// TIA Portal V17 export
// export: Created 2025-03-10T13:11:22.6633057Z, ExportSetting WithDefaults, DisplayName Totally Integrated Automation Portal, DisplayVersion V17 Update 8, DisplayName TIA Portal Openness, DisplayVersion V17 Update 8, DisplayName TIA Portal Version Control Interface, DisplayVersion V17, DisplayName SINAMICS Startdrive Advanced, DisplayVersion V17 SP2, DisplayName SINAMICS Startdrive G110M, G120, G120C, G120D, G120P, G115D, DisplayVersion V17 SP2, DisplayName SINAMICS Startdrive G130, G150, S120, S150, SINAMICS MV, S210, DisplayVersion V17 SP2, DisplayName STEP 7 Professional, DisplayVersion V17 Update 8, DisplayName SINUMERIK ONE STEP 7 Toolbox, DisplayVersion V17 Update 12, DisplayName SINUMERIK 840D sl STEP 7 Toolbox, DisplayVersion V17 Update 12, DisplayName STEP 7 Safety, DisplayVersion V17 Update 6, DisplayName WinCC Advanced, DisplayVersion V17 Update 8
FUNCTION_BLOCK "FB6600_SAFETY_BRAKE_Z_AXIS"   // FB6600, LAD
{ S7_Optimized_Access := 'FALSE' }
AUTHOR : ETXETAR
VERSION : 1.0
// stored: AutoNumber false, IsIECCheckEnabled false, SetENOAutomatically false, UDAEnableTagReadback false
   VAR_INPUT
      OPTIONS_0 : Byte := 2#0000_0000;   // OPTION
      BLOCKED_1 : Bool;   // BLOCKED INPUT
      UNBLOCKED_1 : Bool;   // UNBLOCKED INPUT
      MAINT_BLOCKED : Bool;   // MAINTENANCE BLOCKED INPUT
      MAINT_UNBLOCKED : Bool;   // MAINTENANCE UNBLOCKED INPUT
      BLOCK_CONDITIONS : Bool;   // BLOCK CONDITIONS INPUT
      UNBLOCK_CONDITIONS : Bool;   // UNBLOCK CONDITIONS INPUT
      AXIS_SELECTED : Bool;   // AXES SCREEN AXIS SELECTED
      TRAVERSE_COMMAND : Bool;   // TRAVERSE COMMAND FOR THE AXIS
      UNBLOCK_MAN_REQUEST : Bool;   // UNBLOCK MANUAL REQUEST
      BLOCK_AUTO_REQUEST : Bool;   // BLOCK AUTO REQUEST
      UNBLOCK_AUTO_REQUEST : Bool;   // UNBLOCK AUTO REQUEST
      BRAKE_TEST : Bool;   // BRAKE TEST SIGNAL OF THE AXIS
      UNIT_ALARM : UInt;   // UNIT NUMBER MAX. NUMBER=10
      STATION_ALARM : UInt;   // UNIT NUMBER MAX. NUMBER=10
   END_VAR
   VAR_OUTPUT
      BLOCKED : Bool;   // BLOCKED
      UNBLOCKED : Bool;   // UNBLOCKED
      BLOCKED_ALARM : Bool;   // BLOCKED ALARM
      UNBLOCKED_ALARM : Bool;   // UNBLOCKED ALARM
      MAINTENANCE_UNBLOCKED_ALARM : Bool;   // MAINTENANCE UNBLOCKED ALARM
      BLOCK : Bool;   // BLOCK
      UNBLOCK : Bool;   // UNBLOCK
   END_VAR
   VAR DB_SPECIFIC
      BRAKE { S7_SetPoint := 'True'} : "SAFETY_BRAKE";
      TIMER_BLOCKED { S7_SetPoint := 'True'} : TON_TIME;   // BLOCKED TIMER
      TIMER_UNBLOCKED { S7_SetPoint := 'True'} : TON_TIME;   // UNBLOCKED TIMER
      TIMER_SIMULTANEITY { S7_SetPoint := 'True'} : TON_TIME;   // SIMULTANEITY TIMER
      TIMER_TIME_EXCEEDED { S7_SetPoint := 'True'} : TON_TIME;   // TIME EXCEEDED TIMER
   END_VAR
   VAR_TEMP
      INPUTS_MASK : Byte;   // INPUT MASK
      O_BYTE_0 : Struct   // OPTIONS BYTE 0
         MAINTENANCE_SENSORS : Bool;   // MAINTENANCE SENSORS OPTION
         SPARE_1 : Bool;   // SPARE OPTION
         SPARE_2 : Bool;   // SPARE OPTION
         SPARE_3 : Bool;   // SPARE OPTION
         SPARE_4 : Bool;   // SPARE OPTION
         SPARE_5 : Bool;   // SPARE OPTION
         SPARE_6 : Bool;   // SPARE OPTION
         SPARE_7 : Bool;   // SPARE OPTION
      END_STRUCT;
      DB_NUMBER : DInt;   // DB NUMBER FOR ALARM AND HELP DECODING
   END_VAR
   // TIMER_BLOCKED.PT := T#200ms;
   // TIMER_UNBLOCKED.PT := T#150ms;
   // TIMER_SIMULTANEITY.PT := T#20ms;
   // TIMER_TIME_EXCEEDED.PT := T#2S;
   VAR_TEMP   // added for the SCL form of the ladder/FBD networks
      _w1 : Bool;
      _w2 : Bool;
   END_VAR
BEGIN

NETWORK
TITLE = READ INSTANCE DB
      L     DINO;
      +     10#800000;
      T     #DB_NUMBER;


REGION Network 2: OPTIONS
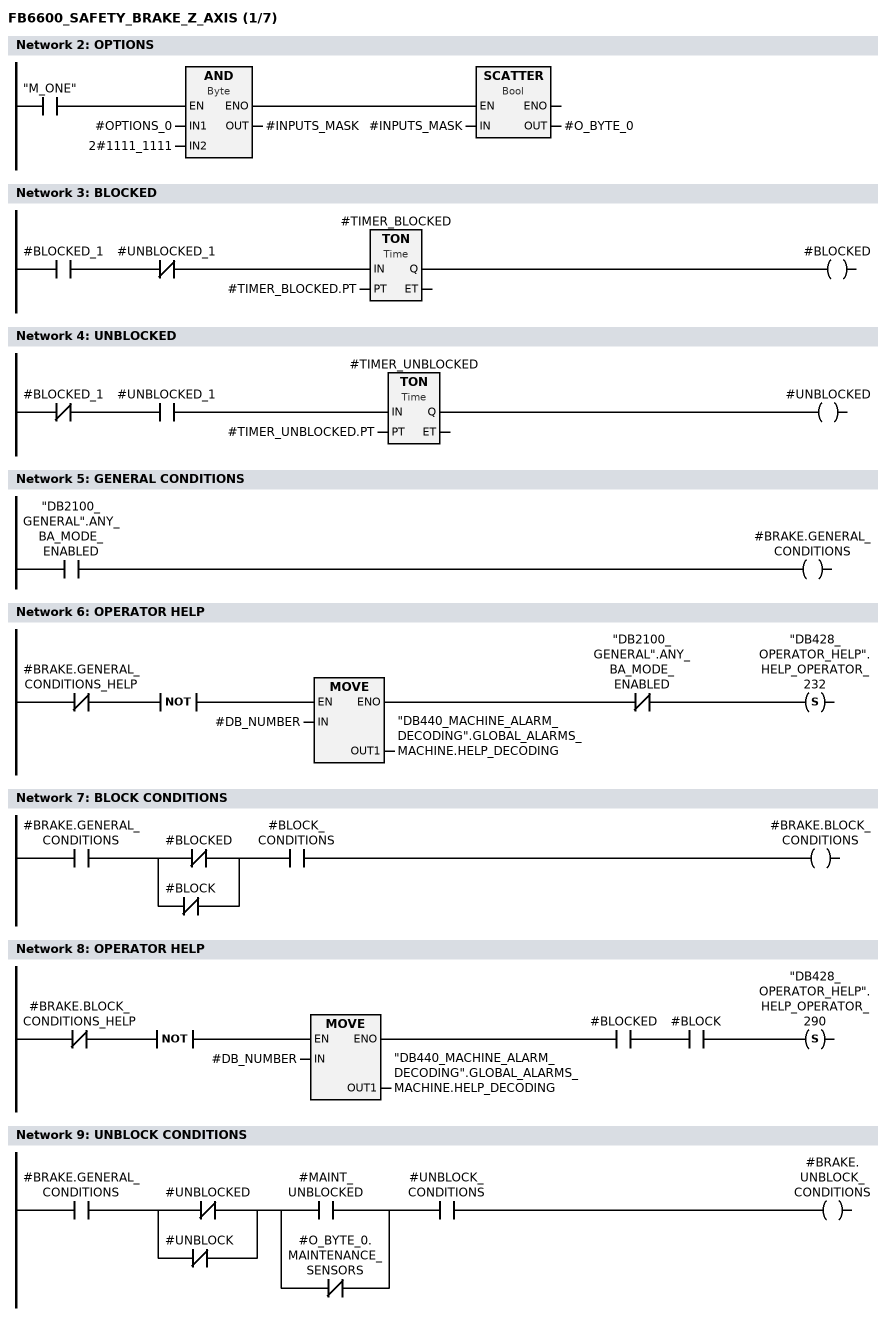
   RUNG wire#powerrail
      Contact( "M_ONE" )
      { S7_Templates := "SrcType := Byte"; S7_GenerateENO := "TRUE" } And(in1 := #OPTIONS_0, in2 := 2#1111_1111, out => #INPUTS_MASK)
      { S7_Templates := "[dest_type := Bool, src_type := Byte]" } SCATTER(IN := #INPUTS_MASK, OUT => #O_BYTE_0)
   END_RUNG
   // the same network as SCL:
   IF "M_ONE" THEN
       #INPUTS_MASK := #OPTIONS_0 AND 2#1111_1111;
       SCATTER(IN := #INPUTS_MASK, OUT => #O_BYTE_0);
   END_IF;
END_REGION

REGION Network 3: BLOCKED
   RUNG wire#powerrail
      Contact( #BLOCKED_1 )
      I_Contact( #UNBLOCKED_1 )
      { S7_Templates := "time_type := Time" } #TIMER_BLOCKED.TON(pt := #TIMER_BLOCKED.PT, et =>)
      Coil( #BLOCKED )
   END_RUNG
   // the same network as SCL:
   #TIMER_BLOCKED(IN := #BLOCKED_1 AND NOT #UNBLOCKED_1, PT := #TIMER_BLOCKED.PT);   // TON
   #BLOCKED := #TIMER_BLOCKED.Q;
END_REGION

REGION Network 4: UNBLOCKED
   RUNG wire#powerrail
      I_Contact( #BLOCKED_1 )
      Contact( #UNBLOCKED_1 )
      { S7_Templates := "time_type := Time" } #TIMER_UNBLOCKED.TON(pt := #TIMER_UNBLOCKED.PT, et =>)
      Coil( #UNBLOCKED )
   END_RUNG
   // the same network as SCL:
   #TIMER_UNBLOCKED(IN := NOT #BLOCKED_1 AND #UNBLOCKED_1, PT := #TIMER_UNBLOCKED.PT);   // TON
   #UNBLOCKED := #TIMER_UNBLOCKED.Q;
END_REGION

REGION Network 5: GENERAL CONDITIONS
   RUNG wire#powerrail
      Contact( "DB2100_GENERAL".ANY_BA_MODE_ENABLED )
      Coil( #BRAKE.GENERAL_CONDITIONS )
   END_RUNG
   // the same network as SCL:
   #BRAKE.GENERAL_CONDITIONS := "DB2100_GENERAL".ANY_BA_MODE_ENABLED;
END_REGION

REGION Network 6: OPERATOR HELP
   RUNG wire#powerrail
      I_Contact( #BRAKE.GENERAL_CONDITIONS_HELP )
      Not()
      { S7_GenerateENO := "TRUE" } Move(in := #DB_NUMBER, out1 => "DB440_MACHINE_ALARM_DECODING".GLOBAL_ALARMS_MACHINE.HELP_DECODING)
      I_Contact( "DB2100_GENERAL".ANY_BA_MODE_ENABLED )
      S_Coil( "DB428_OPERATOR_HELP".HELP_OPERATOR_232 )
   END_RUNG
   // the same network as SCL:
   // ENO of a box is taken as its EN; it also drops when the box reports an error
   #_w1 := NOT (NOT #BRAKE.GENERAL_CONDITIONS_HELP);
   IF #_w1 THEN "DB440_MACHINE_ALARM_DECODING".GLOBAL_ALARMS_MACHINE.HELP_DECODING := #DB_NUMBER; END_IF;
   IF #_w1 AND NOT "DB2100_GENERAL".ANY_BA_MODE_ENABLED THEN
       "DB428_OPERATOR_HELP".HELP_OPERATOR_232 := TRUE;
   END_IF;
END_REGION

REGION Network 7: BLOCK CONDITIONS
   RUNG wire#powerrail
      Contact( #BRAKE.GENERAL_CONDITIONS )
      wire#w1
      I_Contact( #BLOCKED )
      wire#w2
      Contact( #BLOCK_CONDITIONS )
      Coil( #BRAKE.BLOCK_CONDITIONS )
   END_RUNG
   RUNG wire#w1
      I_Contact( #BLOCK )
   END_RUNG wire#w2
   // the same network as SCL:
   #BRAKE.BLOCK_CONDITIONS := #BRAKE.GENERAL_CONDITIONS AND (NOT #BLOCKED OR NOT #BLOCK) AND #BLOCK_CONDITIONS;
END_REGION

REGION Network 8: OPERATOR HELP
   RUNG wire#powerrail
      I_Contact( #BRAKE.BLOCK_CONDITIONS_HELP )
      Not()
      { S7_GenerateENO := "TRUE" } Move(in := #DB_NUMBER, out1 => "DB440_MACHINE_ALARM_DECODING".GLOBAL_ALARMS_MACHINE.HELP_DECODING)
      Contact( #BLOCKED )
      Contact( #BLOCK )
      S_Coil( "DB428_OPERATOR_HELP".HELP_OPERATOR_290 )
   END_RUNG
   // the same network as SCL:
   // ENO of a box is taken as its EN; it also drops when the box reports an error
   #_w1 := NOT (NOT #BRAKE.BLOCK_CONDITIONS_HELP);
   IF #_w1 THEN "DB440_MACHINE_ALARM_DECODING".GLOBAL_ALARMS_MACHINE.HELP_DECODING := #DB_NUMBER; END_IF;
   IF #_w1 AND #BLOCKED AND #BLOCK THEN "DB428_OPERATOR_HELP".HELP_OPERATOR_290 := TRUE; END_IF;
END_REGION

REGION Network 9: UNBLOCK CONDITIONS
   RUNG wire#powerrail
      Contact( #BRAKE.GENERAL_CONDITIONS )
      wire#w1
      I_Contact( #UNBLOCKED )
      wire#w2
      Contact( #MAINT_UNBLOCKED )
      wire#w3
      Contact( #UNBLOCK_CONDITIONS )
      Coil( #BRAKE.UNBLOCK_CONDITIONS )
   END_RUNG
   RUNG wire#w1
      I_Contact( #UNBLOCK )
   END_RUNG wire#w2
   RUNG wire#w2
      I_Contact( #O_BYTE_0.MAINTENANCE_SENSORS )
   END_RUNG wire#w3
   // the same network as SCL:
   #BRAKE.UNBLOCK_CONDITIONS := #BRAKE.GENERAL_CONDITIONS AND (NOT #UNBLOCKED OR NOT #UNBLOCK) AND (#MAINT_UNBLOCKED OR NOT #O_BYTE_0.MAINTENANCE_SENSORS) AND #UNBLOCK_CONDITIONS;
END_REGION

REGION Network 10: OPERATOR HELP
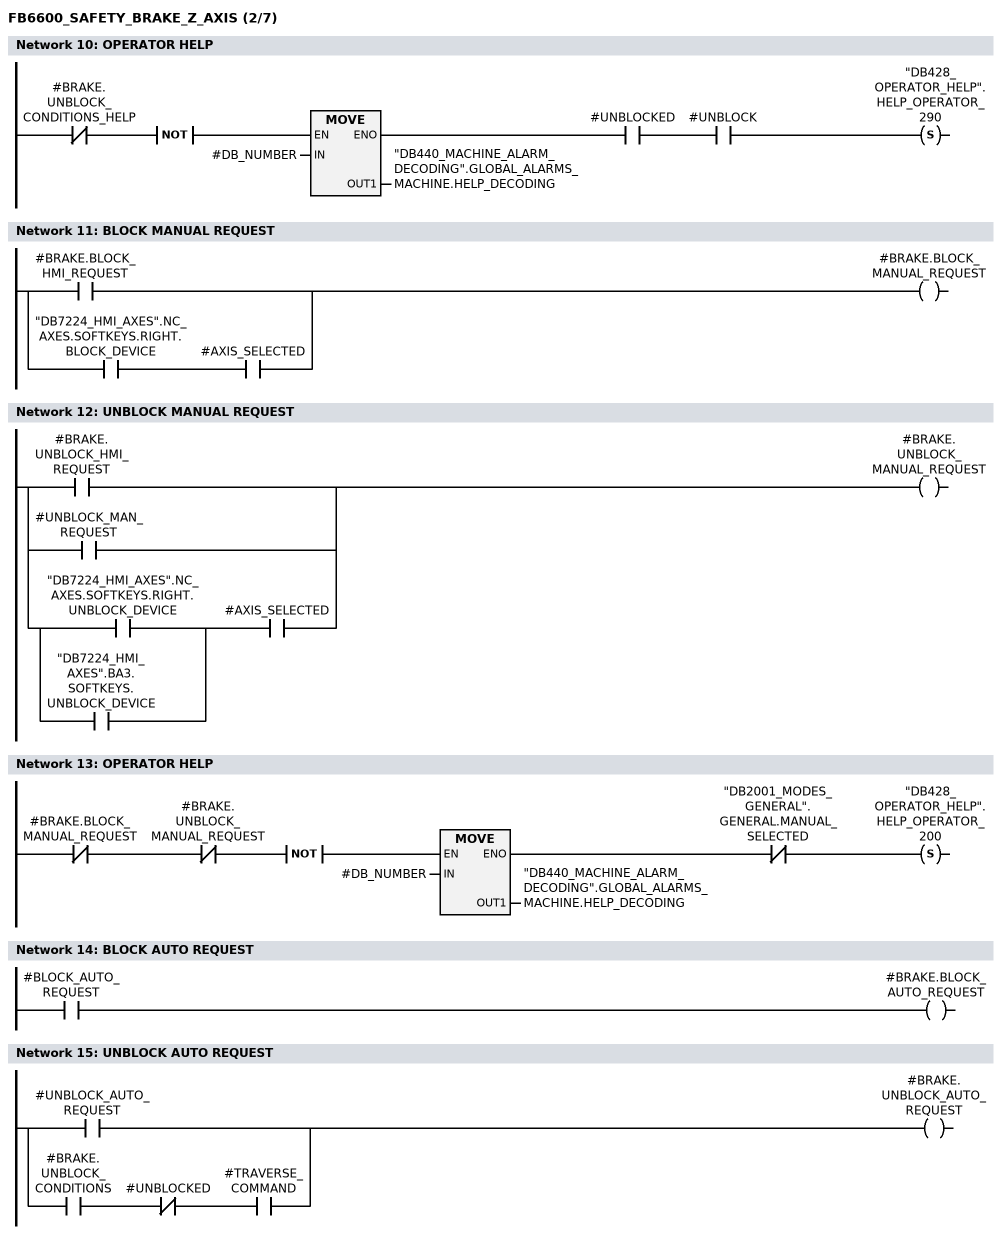
   RUNG wire#powerrail
      I_Contact( #BRAKE.UNBLOCK_CONDITIONS_HELP )
      Not()
      { S7_GenerateENO := "TRUE" } Move(in := #DB_NUMBER, out1 => "DB440_MACHINE_ALARM_DECODING".GLOBAL_ALARMS_MACHINE.HELP_DECODING)
      Contact( #UNBLOCKED )
      Contact( #UNBLOCK )
      S_Coil( "DB428_OPERATOR_HELP".HELP_OPERATOR_290 )
   END_RUNG
   // the same network as SCL:
   // ENO of a box is taken as its EN; it also drops when the box reports an error
   #_w1 := NOT (NOT #BRAKE.UNBLOCK_CONDITIONS_HELP);
   IF #_w1 THEN "DB440_MACHINE_ALARM_DECODING".GLOBAL_ALARMS_MACHINE.HELP_DECODING := #DB_NUMBER; END_IF;
   IF #_w1 AND #UNBLOCKED AND #UNBLOCK THEN "DB428_OPERATOR_HELP".HELP_OPERATOR_290 := TRUE; END_IF;
END_REGION

REGION Network 11: BLOCK MANUAL REQUEST
   RUNG wire#powerrail
      Contact( #BRAKE.BLOCK_HMI_REQUEST )
      wire#w1
      Coil( #BRAKE.BLOCK_MANUAL_REQUEST )
   END_RUNG
   RUNG wire#powerrail
      Contact( "DB7224_HMI_AXES".NC_AXES.SOFTKEYS.RIGHT.BLOCK_DEVICE )
      Contact( #AXIS_SELECTED )
   END_RUNG wire#w1
   // the same network as SCL:
   #BRAKE.BLOCK_MANUAL_REQUEST := #BRAKE.BLOCK_HMI_REQUEST OR ("DB7224_HMI_AXES".NC_AXES.SOFTKEYS.RIGHT.BLOCK_DEVICE AND #AXIS_SELECTED);
END_REGION

REGION Network 12: UNBLOCK MANUAL REQUEST
   RUNG wire#powerrail
      Contact( #BRAKE.UNBLOCK_HMI_REQUEST )
      wire#w1
      Coil( #BRAKE.UNBLOCK_MANUAL_REQUEST )
   END_RUNG
   RUNG wire#powerrail
      Contact( #UNBLOCK_MAN_REQUEST )
   END_RUNG wire#w1
   RUNG wire#powerrail
      Contact( "DB7224_HMI_AXES".NC_AXES.SOFTKEYS.RIGHT.UNBLOCK_DEVICE )
      wire#w2
      Contact( #AXIS_SELECTED )
   END_RUNG wire#w1
   RUNG wire#powerrail
      Contact( "DB7224_HMI_AXES".BA3.SOFTKEYS.UNBLOCK_DEVICE )
   END_RUNG wire#w2
   // the same network as SCL:
   #BRAKE.UNBLOCK_MANUAL_REQUEST := #BRAKE.UNBLOCK_HMI_REQUEST OR #UNBLOCK_MAN_REQUEST OR (("DB7224_HMI_AXES".NC_AXES.SOFTKEYS.RIGHT.UNBLOCK_DEVICE OR "DB7224_HMI_AXES".BA3.SOFTKEYS.UNBLOCK_DEVICE) AND #AXIS_SELECTED);
END_REGION

REGION Network 13: OPERATOR HELP
   RUNG wire#powerrail
      I_Contact( #BRAKE.BLOCK_MANUAL_REQUEST )
      I_Contact( #BRAKE.UNBLOCK_MANUAL_REQUEST )
      Not()
      { S7_GenerateENO := "TRUE" } Move(in := #DB_NUMBER, out1 => "DB440_MACHINE_ALARM_DECODING".GLOBAL_ALARMS_MACHINE.HELP_DECODING)
      I_Contact( "DB2001_MODES_GENERAL".GENERAL.MANUAL_SELECTED )
      S_Coil( "DB428_OPERATOR_HELP".HELP_OPERATOR_200 )
   END_RUNG
   // the same network as SCL:
   // ENO of a box is taken as its EN; it also drops when the box reports an error
   #_w1 := NOT (NOT #BRAKE.BLOCK_MANUAL_REQUEST AND NOT #BRAKE.UNBLOCK_MANUAL_REQUEST);
   IF #_w1 THEN "DB440_MACHINE_ALARM_DECODING".GLOBAL_ALARMS_MACHINE.HELP_DECODING := #DB_NUMBER; END_IF;
   IF #_w1 AND NOT "DB2001_MODES_GENERAL".GENERAL.MANUAL_SELECTED THEN
       "DB428_OPERATOR_HELP".HELP_OPERATOR_200 := TRUE;
   END_IF;
END_REGION

REGION Network 14: BLOCK AUTO REQUEST
   RUNG wire#powerrail
      Contact( #BLOCK_AUTO_REQUEST )
      Coil( #BRAKE.BLOCK_AUTO_REQUEST )
   END_RUNG
   // the same network as SCL:
   #BRAKE.BLOCK_AUTO_REQUEST := #BLOCK_AUTO_REQUEST;
END_REGION

REGION Network 15: UNBLOCK AUTO REQUEST
   RUNG wire#powerrail
      Contact( #UNBLOCK_AUTO_REQUEST )
      wire#w1
      Coil( #BRAKE.UNBLOCK_AUTO_REQUEST )
   END_RUNG
   RUNG wire#powerrail
      Contact( #BRAKE.UNBLOCK_CONDITIONS )
      I_Contact( #UNBLOCKED )
      Contact( #TRAVERSE_COMMAND )
   END_RUNG wire#w1
   // the same network as SCL:
   #BRAKE.UNBLOCK_AUTO_REQUEST := #UNBLOCK_AUTO_REQUEST OR (#BRAKE.UNBLOCK_CONDITIONS AND NOT #UNBLOCKED AND #TRAVERSE_COMMAND);
END_REGION

REGION Network 16: BLOCK GLOBAL REQUEST
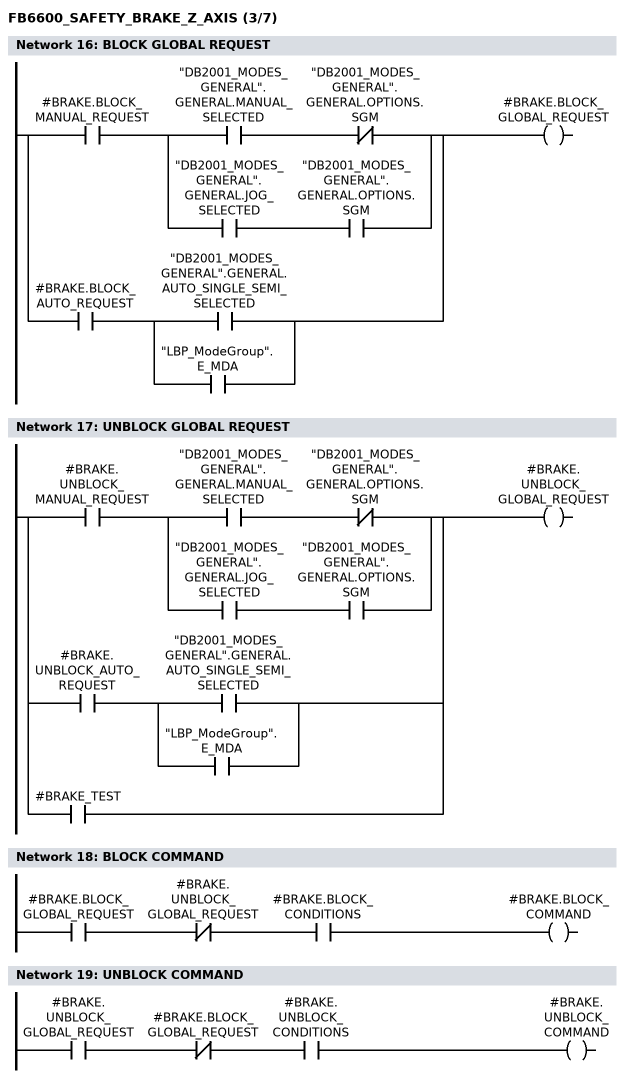
   RUNG wire#powerrail
      Contact( #BRAKE.BLOCK_MANUAL_REQUEST )
      wire#w1
      Contact( "DB2001_MODES_GENERAL".GENERAL.MANUAL_SELECTED )
      I_Contact( "DB2001_MODES_GENERAL".GENERAL.OPTIONS.SGM )
      wire#w2
      Coil( #BRAKE.BLOCK_GLOBAL_REQUEST )
   END_RUNG
   RUNG wire#w1
      Contact( "DB2001_MODES_GENERAL".GENERAL.JOG_SELECTED )
      Contact( "DB2001_MODES_GENERAL".GENERAL.OPTIONS.SGM )
   END_RUNG wire#w2
   RUNG wire#powerrail
      Contact( #BRAKE.BLOCK_AUTO_REQUEST )
      wire#w3
      Contact( "DB2001_MODES_GENERAL".GENERAL.AUTO_SINGLE_SEMI_SELECTED )
   END_RUNG wire#w2
   RUNG wire#w3
      Contact( "LBP_ModeGroup".E_MDA )
   END_RUNG wire#w2
   // the same network as SCL:
   #BRAKE.BLOCK_GLOBAL_REQUEST := (#BRAKE.BLOCK_MANUAL_REQUEST AND (("DB2001_MODES_GENERAL".GENERAL.MANUAL_SELECTED AND NOT "DB2001_MODES_GENERAL".GENERAL.OPTIONS.SGM) OR ("DB2001_MODES_GENERAL".GENERAL.JOG_SELECTED AND "DB2001_MODES_GENERAL".GENERAL.OPTIONS.SGM))) OR (#BRAKE.BLOCK_AUTO_REQUEST AND ("DB2001_MODES_GENERAL".GENERAL.AUTO_SINGLE_SEMI_SELECTED OR "LBP_ModeGroup".E_MDA));
END_REGION

REGION Network 17: UNBLOCK GLOBAL REQUEST
   RUNG wire#powerrail
      Contact( #BRAKE.UNBLOCK_MANUAL_REQUEST )
      wire#w1
      Contact( "DB2001_MODES_GENERAL".GENERAL.MANUAL_SELECTED )
      I_Contact( "DB2001_MODES_GENERAL".GENERAL.OPTIONS.SGM )
      wire#w2
      Coil( #BRAKE.UNBLOCK_GLOBAL_REQUEST )
   END_RUNG
   RUNG wire#w1
      Contact( "DB2001_MODES_GENERAL".GENERAL.JOG_SELECTED )
      Contact( "DB2001_MODES_GENERAL".GENERAL.OPTIONS.SGM )
   END_RUNG wire#w2
   RUNG wire#powerrail
      Contact( #BRAKE.UNBLOCK_AUTO_REQUEST )
      wire#w3
      Contact( "DB2001_MODES_GENERAL".GENERAL.AUTO_SINGLE_SEMI_SELECTED )
   END_RUNG wire#w2
   RUNG wire#w3
      Contact( "LBP_ModeGroup".E_MDA )
   END_RUNG wire#w2
   RUNG wire#powerrail
      Contact( #BRAKE_TEST )
   END_RUNG wire#w2
   // the same network as SCL:
   #BRAKE.UNBLOCK_GLOBAL_REQUEST := (#BRAKE.UNBLOCK_MANUAL_REQUEST AND (("DB2001_MODES_GENERAL".GENERAL.MANUAL_SELECTED AND NOT "DB2001_MODES_GENERAL".GENERAL.OPTIONS.SGM) OR ("DB2001_MODES_GENERAL".GENERAL.JOG_SELECTED AND "DB2001_MODES_GENERAL".GENERAL.OPTIONS.SGM))) OR (#BRAKE.UNBLOCK_AUTO_REQUEST AND ("DB2001_MODES_GENERAL".GENERAL.AUTO_SINGLE_SEMI_SELECTED OR "LBP_ModeGroup".E_MDA)) OR #BRAKE_TEST;
END_REGION

REGION Network 18: BLOCK COMMAND
   RUNG wire#powerrail
      Contact( #BRAKE.BLOCK_GLOBAL_REQUEST )
      I_Contact( #BRAKE.UNBLOCK_GLOBAL_REQUEST )
      Contact( #BRAKE.BLOCK_CONDITIONS )
      Coil( #BRAKE.BLOCK_COMMAND )
   END_RUNG
   // the same network as SCL:
   #BRAKE.BLOCK_COMMAND := #BRAKE.BLOCK_GLOBAL_REQUEST AND NOT #BRAKE.UNBLOCK_GLOBAL_REQUEST AND #BRAKE.BLOCK_CONDITIONS;
END_REGION

REGION Network 19: UNBLOCK COMMAND
   RUNG wire#powerrail
      Contact( #BRAKE.UNBLOCK_GLOBAL_REQUEST )
      I_Contact( #BRAKE.BLOCK_GLOBAL_REQUEST )
      Contact( #BRAKE.UNBLOCK_CONDITIONS )
      Coil( #BRAKE.UNBLOCK_COMMAND )
   END_RUNG
   // the same network as SCL:
   #BRAKE.UNBLOCK_COMMAND := #BRAKE.UNBLOCK_GLOBAL_REQUEST AND NOT #BRAKE.BLOCK_GLOBAL_REQUEST AND #BRAKE.UNBLOCK_CONDITIONS;
END_REGION

REGION Network 20: BLOCK
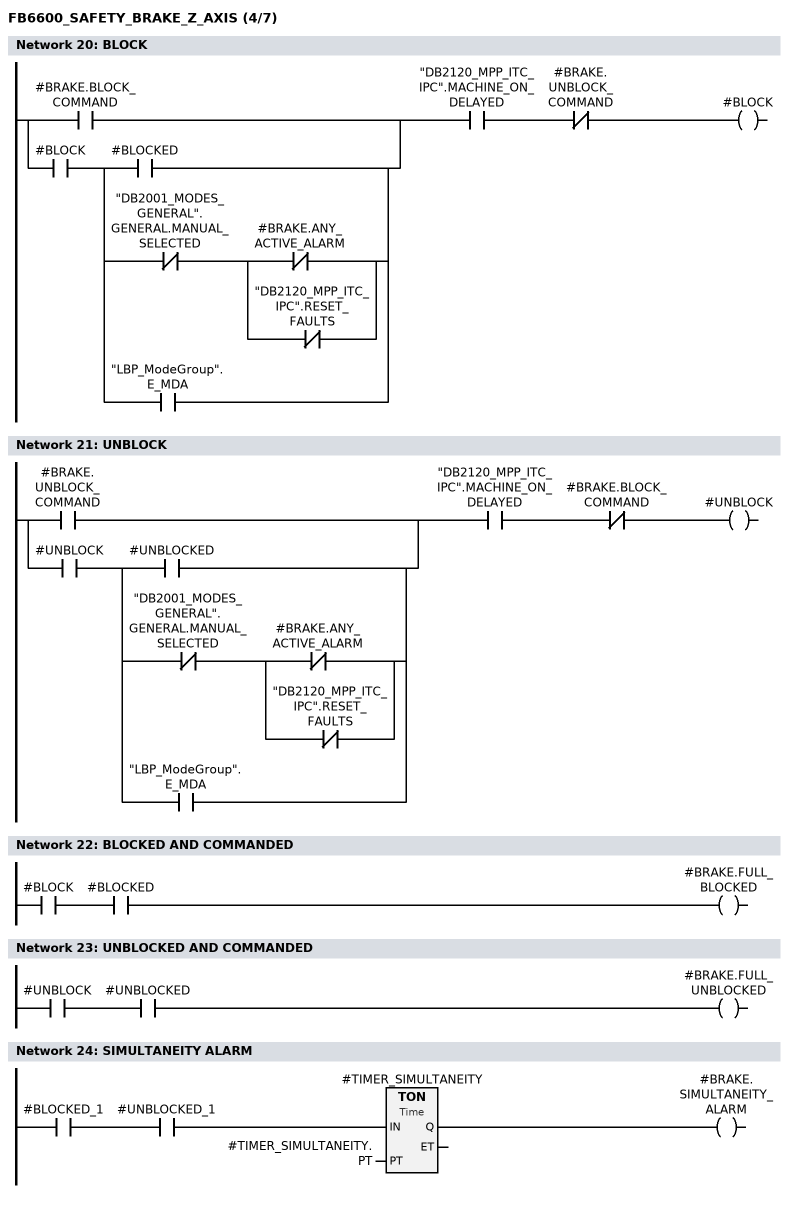
   RUNG wire#powerrail
      Contact( #BRAKE.BLOCK_COMMAND )
      wire#w1
      Contact( "DB2120_MPP_ITC_IPC".MACHINE_ON_DELAYED )
      I_Contact( #BRAKE.UNBLOCK_COMMAND )
      Coil( #BLOCK )
   END_RUNG
   RUNG wire#powerrail
      Contact( #BLOCK )
      wire#w2
      Contact( #BLOCKED )
   END_RUNG wire#w1
   RUNG wire#w2
      I_Contact( "DB2001_MODES_GENERAL".GENERAL.MANUAL_SELECTED )
      wire#w3
      I_Contact( #BRAKE.ANY_ACTIVE_ALARM )
   END_RUNG wire#w1
   RUNG wire#w3
      I_Contact( "DB2120_MPP_ITC_IPC".RESET_FAULTS )
   END_RUNG wire#w1
   RUNG wire#w2
      Contact( "LBP_ModeGroup".E_MDA )
   END_RUNG wire#w1
   // the same network as SCL:
   #BLOCK := (#BRAKE.BLOCK_COMMAND OR (#BLOCK AND (#BLOCKED OR (NOT "DB2001_MODES_GENERAL".GENERAL.MANUAL_SELECTED AND (NOT #BRAKE.ANY_ACTIVE_ALARM OR NOT "DB2120_MPP_ITC_IPC".RESET_FAULTS)) OR "LBP_ModeGroup".E_MDA))) AND "DB2120_MPP_ITC_IPC".MACHINE_ON_DELAYED AND NOT #BRAKE.UNBLOCK_COMMAND;
END_REGION

REGION Network 21: UNBLOCK
   RUNG wire#powerrail
      Contact( #BRAKE.UNBLOCK_COMMAND )
      wire#w1
      Contact( "DB2120_MPP_ITC_IPC".MACHINE_ON_DELAYED )
      I_Contact( #BRAKE.BLOCK_COMMAND )
      Coil( #UNBLOCK )
   END_RUNG
   RUNG wire#powerrail
      Contact( #UNBLOCK )
      wire#w2
      Contact( #UNBLOCKED )
   END_RUNG wire#w1
   RUNG wire#w2
      I_Contact( "DB2001_MODES_GENERAL".GENERAL.MANUAL_SELECTED )
      wire#w3
      I_Contact( #BRAKE.ANY_ACTIVE_ALARM )
   END_RUNG wire#w1
   RUNG wire#w3
      I_Contact( "DB2120_MPP_ITC_IPC".RESET_FAULTS )
   END_RUNG wire#w1
   RUNG wire#w2
      Contact( "LBP_ModeGroup".E_MDA )
   END_RUNG wire#w1
   // the same network as SCL:
   #UNBLOCK := (#BRAKE.UNBLOCK_COMMAND OR (#UNBLOCK AND (#UNBLOCKED OR (NOT "DB2001_MODES_GENERAL".GENERAL.MANUAL_SELECTED AND (NOT #BRAKE.ANY_ACTIVE_ALARM OR NOT "DB2120_MPP_ITC_IPC".RESET_FAULTS)) OR "LBP_ModeGroup".E_MDA))) AND "DB2120_MPP_ITC_IPC".MACHINE_ON_DELAYED AND NOT #BRAKE.BLOCK_COMMAND;
END_REGION

REGION Network 22: BLOCKED AND COMMANDED
   RUNG wire#powerrail
      Contact( #BLOCK )
      Contact( #BLOCKED )
      Coil( #BRAKE.FULL_BLOCKED )
   END_RUNG
   // the same network as SCL:
   #BRAKE.FULL_BLOCKED := #BLOCK AND #BLOCKED;
END_REGION

REGION Network 23: UNBLOCKED AND COMMANDED
   RUNG wire#powerrail
      Contact( #UNBLOCK )
      Contact( #UNBLOCKED )
      Coil( #BRAKE.FULL_UNBLOCKED )
   END_RUNG
   // the same network as SCL:
   #BRAKE.FULL_UNBLOCKED := #UNBLOCK AND #UNBLOCKED;
END_REGION

REGION Network 24: SIMULTANEITY ALARM
   RUNG wire#powerrail
      Contact( #BLOCKED_1 )
      Contact( #UNBLOCKED_1 )
      { S7_Templates := "time_type := Time" } #TIMER_SIMULTANEITY.TON(pt := #TIMER_SIMULTANEITY.PT, et =>)
      Coil( #BRAKE.SIMULTANEITY_ALARM )
   END_RUNG
   // the same network as SCL:
   #TIMER_SIMULTANEITY(IN := #BLOCKED_1 AND #UNBLOCKED_1, PT := #TIMER_SIMULTANEITY.PT);   // TON
   #BRAKE.SIMULTANEITY_ALARM := #TIMER_SIMULTANEITY.Q;
END_REGION

REGION Network 25: TIME EXCEEDED ALARM
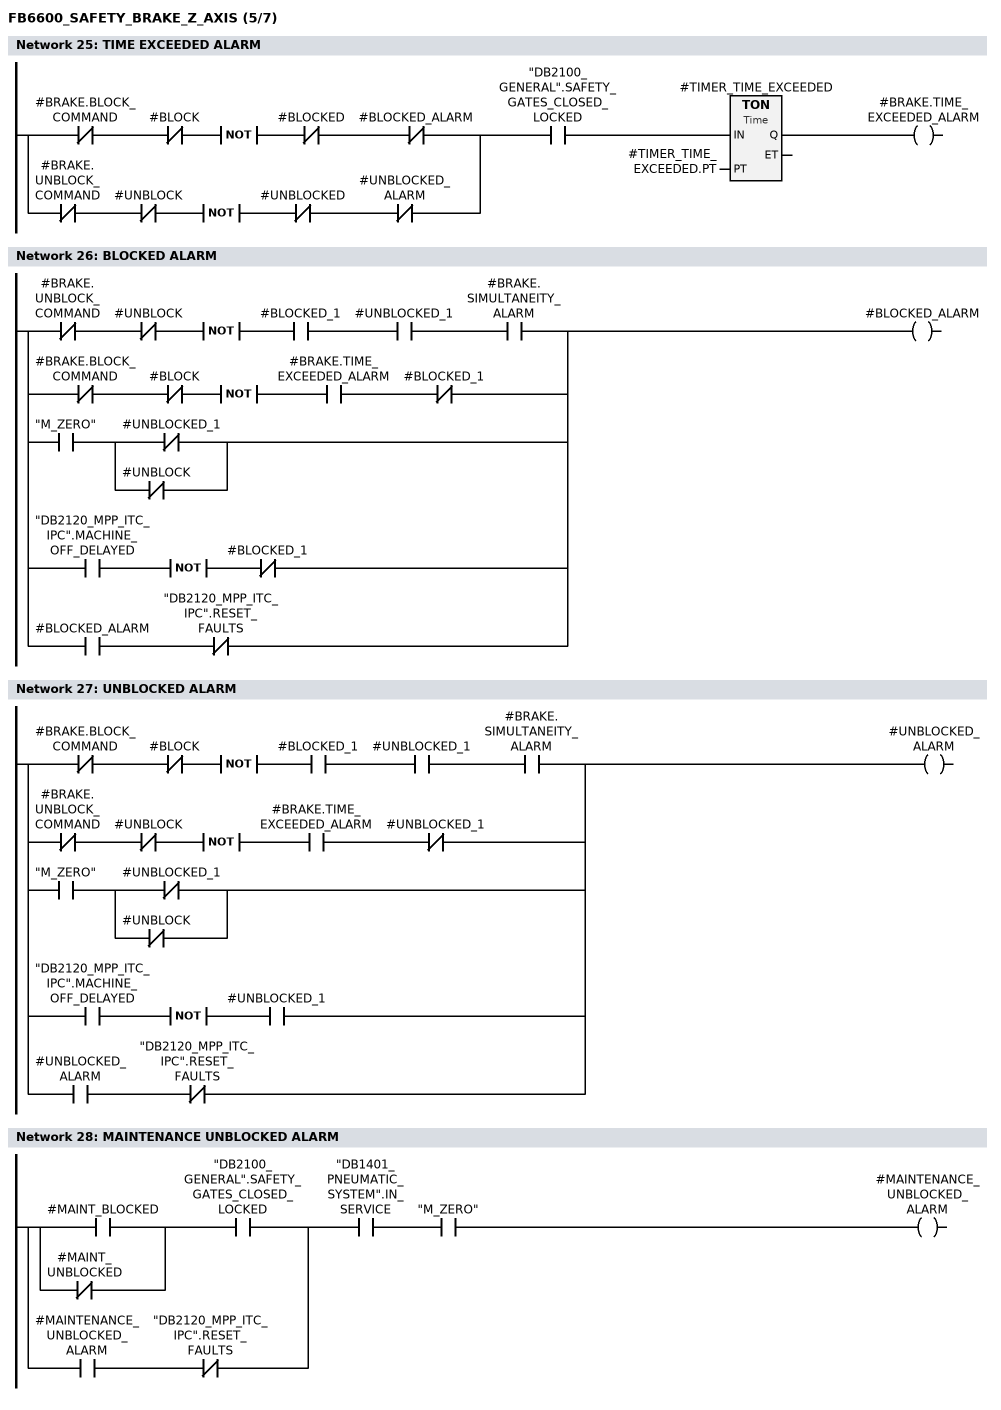
   RUNG wire#powerrail
      I_Contact( #BRAKE.BLOCK_COMMAND )
      I_Contact( #BLOCK )
      Not()
      I_Contact( #BLOCKED )
      I_Contact( #BLOCKED_ALARM )
      wire#w1
      Contact( "DB2100_GENERAL".SAFETY_GATES_CLOSED_LOCKED )
      { S7_Templates := "time_type := Time" } #TIMER_TIME_EXCEEDED.TON(pt := #TIMER_TIME_EXCEEDED.PT, et =>)
      Coil( #BRAKE.TIME_EXCEEDED_ALARM )
   END_RUNG
   RUNG wire#powerrail
      I_Contact( #BRAKE.UNBLOCK_COMMAND )
      I_Contact( #UNBLOCK )
      Not()
      I_Contact( #UNBLOCKED )
      I_Contact( #UNBLOCKED_ALARM )
   END_RUNG wire#w1
   // the same network as SCL:
   #TIMER_TIME_EXCEEDED(IN := ((NOT (NOT #BRAKE.BLOCK_COMMAND AND NOT #BLOCK) AND NOT #BLOCKED AND NOT #BLOCKED_ALARM) OR (NOT (NOT #BRAKE.UNBLOCK_COMMAND AND NOT #UNBLOCK) AND NOT #UNBLOCKED AND NOT #UNBLOCKED_ALARM)) AND "DB2100_GENERAL".SAFETY_GATES_CLOSED_LOCKED,   // TON
                        PT := #TIMER_TIME_EXCEEDED.PT);
   #BRAKE.TIME_EXCEEDED_ALARM := #TIMER_TIME_EXCEEDED.Q;
END_REGION

REGION Network 26: BLOCKED ALARM
   RUNG wire#powerrail
      I_Contact( #BRAKE.UNBLOCK_COMMAND )
      I_Contact( #UNBLOCK )
      Not()
      Contact( #BLOCKED_1 )
      Contact( #UNBLOCKED_1 )
      Contact( #BRAKE.SIMULTANEITY_ALARM )
      wire#w1
      Coil( #BLOCKED_ALARM )
   END_RUNG
   RUNG wire#powerrail
      I_Contact( #BRAKE.BLOCK_COMMAND )
      I_Contact( #BLOCK )
      Not()
      Contact( #BRAKE.TIME_EXCEEDED_ALARM )
      I_Contact( #BLOCKED_1 )
   END_RUNG wire#w1
   RUNG wire#powerrail
      Contact( "M_ZERO" )
      wire#w2
      I_Contact( #UNBLOCKED_1 )
   END_RUNG wire#w1
   RUNG wire#w2
      I_Contact( #UNBLOCK )
   END_RUNG wire#w1
   RUNG wire#powerrail
      Contact( "DB2120_MPP_ITC_IPC".MACHINE_OFF_DELAYED )
      Not()
      I_Contact( #BLOCKED_1 )
   END_RUNG wire#w1
   RUNG wire#powerrail
      Contact( #BLOCKED_ALARM )
      I_Contact( "DB2120_MPP_ITC_IPC".RESET_FAULTS )
   END_RUNG wire#w1
   // the same network as SCL:
   #BLOCKED_ALARM := (NOT (NOT #BRAKE.UNBLOCK_COMMAND AND NOT #UNBLOCK) AND #BLOCKED_1 AND #UNBLOCKED_1 AND #BRAKE.SIMULTANEITY_ALARM) OR (NOT (NOT #BRAKE.BLOCK_COMMAND AND NOT #BLOCK) AND #BRAKE.TIME_EXCEEDED_ALARM AND NOT #BLOCKED_1) OR ("M_ZERO" AND (NOT #UNBLOCKED_1 OR NOT #UNBLOCK)) OR (NOT "DB2120_MPP_ITC_IPC".MACHINE_OFF_DELAYED AND NOT #BLOCKED_1) OR (#BLOCKED_ALARM AND NOT "DB2120_MPP_ITC_IPC".RESET_FAULTS);
END_REGION

REGION Network 27: UNBLOCKED ALARM
   RUNG wire#powerrail
      I_Contact( #BRAKE.BLOCK_COMMAND )
      I_Contact( #BLOCK )
      Not()
      Contact( #BLOCKED_1 )
      Contact( #UNBLOCKED_1 )
      Contact( #BRAKE.SIMULTANEITY_ALARM )
      wire#w1
      Coil( #UNBLOCKED_ALARM )
   END_RUNG
   RUNG wire#powerrail
      I_Contact( #BRAKE.UNBLOCK_COMMAND )
      I_Contact( #UNBLOCK )
      Not()
      Contact( #BRAKE.TIME_EXCEEDED_ALARM )
      I_Contact( #UNBLOCKED_1 )
   END_RUNG wire#w1
   RUNG wire#powerrail
      Contact( "M_ZERO" )
      wire#w2
      I_Contact( #UNBLOCKED_1 )
   END_RUNG wire#w1
   RUNG wire#w2
      I_Contact( #UNBLOCK )
   END_RUNG wire#w1
   RUNG wire#powerrail
      Contact( "DB2120_MPP_ITC_IPC".MACHINE_OFF_DELAYED )
      Not()
      Contact( #UNBLOCKED_1 )
   END_RUNG wire#w1
   RUNG wire#powerrail
      Contact( #UNBLOCKED_ALARM )
      I_Contact( "DB2120_MPP_ITC_IPC".RESET_FAULTS )
   END_RUNG wire#w1
   // the same network as SCL:
   #UNBLOCKED_ALARM := (NOT (NOT #BRAKE.BLOCK_COMMAND AND NOT #BLOCK) AND #BLOCKED_1 AND #UNBLOCKED_1 AND #BRAKE.SIMULTANEITY_ALARM) OR (NOT (NOT #BRAKE.UNBLOCK_COMMAND AND NOT #UNBLOCK) AND #BRAKE.TIME_EXCEEDED_ALARM AND NOT #UNBLOCKED_1) OR ("M_ZERO" AND (NOT #UNBLOCKED_1 OR NOT #UNBLOCK)) OR (NOT "DB2120_MPP_ITC_IPC".MACHINE_OFF_DELAYED AND #UNBLOCKED_1) OR (#UNBLOCKED_ALARM AND NOT "DB2120_MPP_ITC_IPC".RESET_FAULTS);
END_REGION

REGION Network 28: MAINTENANCE UNBLOCKED ALARM
   RUNG wire#powerrail
      Contact( #MAINT_BLOCKED )
      wire#w1
      Contact( "DB2100_GENERAL".SAFETY_GATES_CLOSED_LOCKED )
      wire#w2
      Contact( "DB1401_PNEUMATIC_SYSTEM".IN_SERVICE )
      Contact( "M_ZERO" )
      Coil( #MAINTENANCE_UNBLOCKED_ALARM )
   END_RUNG
   RUNG wire#powerrail
      I_Contact( #MAINT_UNBLOCKED )
   END_RUNG wire#w1
   RUNG wire#powerrail
      Contact( #MAINTENANCE_UNBLOCKED_ALARM )
      I_Contact( "DB2120_MPP_ITC_IPC".RESET_FAULTS )
   END_RUNG wire#w2
   // the same network as SCL:
   #MAINTENANCE_UNBLOCKED_ALARM := (((#MAINT_BLOCKED OR NOT #MAINT_UNBLOCKED) AND "DB2100_GENERAL".SAFETY_GATES_CLOSED_LOCKED) OR (#MAINTENANCE_UNBLOCKED_ALARM AND NOT "DB2120_MPP_ITC_IPC".RESET_FAULTS)) AND "DB1401_PNEUMATIC_SYSTEM".IN_SERVICE AND "M_ZERO";
END_REGION

REGION Network 29: IMMEDIATE STOP AND STOP END OF CYCLE ALARMS
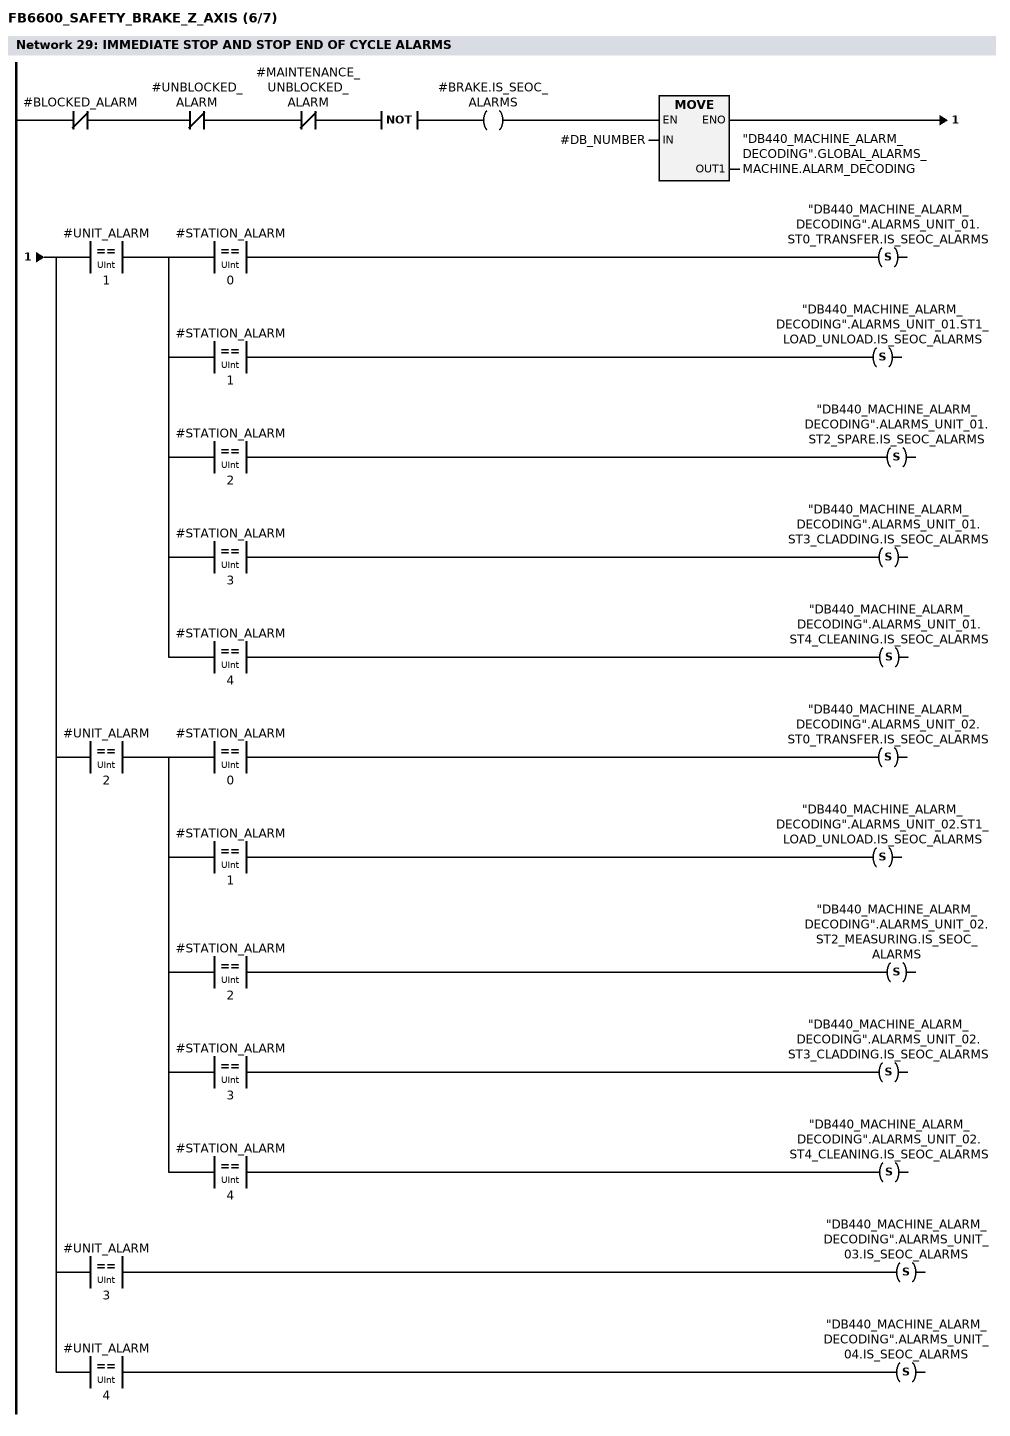
   RUNG wire#powerrail
      I_Contact( #BLOCKED_ALARM )
      I_Contact( #UNBLOCKED_ALARM )
      I_Contact( #MAINTENANCE_UNBLOCKED_ALARM )
      Not()
      Coil( #BRAKE.IS_SEOC_ALARMS )
      { S7_GenerateENO := "TRUE" } Move(in := #DB_NUMBER, out1 => "DB440_MACHINE_ALARM_DECODING".GLOBAL_ALARMS_MACHINE.ALARM_DECODING)
      wire#w1
      { S7_Templates := "SrcType := UInt" } EQ_Contact(in1 := #UNIT_ALARM, in2 := 1)
      wire#w2
      { S7_Templates := "SrcType := UInt" } EQ_Contact(in1 := #STATION_ALARM, in2 := 0)
      S_Coil( "DB440_MACHINE_ALARM_DECODING".ALARMS_UNIT_01.ST0_TRANSFER.IS_SEOC_ALARMS )
   END_RUNG
   RUNG wire#w2
      { S7_Templates := "SrcType := UInt" } EQ_Contact(in1 := #STATION_ALARM, in2 := 1)
      S_Coil( "DB440_MACHINE_ALARM_DECODING".ALARMS_UNIT_01.ST1_LOAD_UNLOAD.IS_SEOC_ALARMS )
   END_RUNG
   RUNG wire#w2
      { S7_Templates := "SrcType := UInt" } EQ_Contact(in1 := #STATION_ALARM, in2 := 2)
      S_Coil( "DB440_MACHINE_ALARM_DECODING".ALARMS_UNIT_01.ST2_SPARE.IS_SEOC_ALARMS )
   END_RUNG
   RUNG wire#w2
      { S7_Templates := "SrcType := UInt" } EQ_Contact(in1 := #STATION_ALARM, in2 := 3)
      S_Coil( "DB440_MACHINE_ALARM_DECODING".ALARMS_UNIT_01.ST3_CLADDING.IS_SEOC_ALARMS )
   END_RUNG
   RUNG wire#w2
      { S7_Templates := "SrcType := UInt" } EQ_Contact(in1 := #STATION_ALARM, in2 := 4)
      S_Coil( "DB440_MACHINE_ALARM_DECODING".ALARMS_UNIT_01.ST4_CLEANING.IS_SEOC_ALARMS )
   END_RUNG
   RUNG wire#w1
      { S7_Templates := "SrcType := UInt" } EQ_Contact(in1 := #UNIT_ALARM, in2 := 2)
      wire#w3
      { S7_Templates := "SrcType := UInt" } EQ_Contact(in1 := #STATION_ALARM, in2 := 0)
      S_Coil( "DB440_MACHINE_ALARM_DECODING".ALARMS_UNIT_02.ST0_TRANSFER.IS_SEOC_ALARMS )
   END_RUNG
   RUNG wire#w3
      { S7_Templates := "SrcType := UInt" } EQ_Contact(in1 := #STATION_ALARM, in2 := 1)
      S_Coil( "DB440_MACHINE_ALARM_DECODING".ALARMS_UNIT_02.ST1_LOAD_UNLOAD.IS_SEOC_ALARMS )
   END_RUNG
   RUNG wire#w3
      { S7_Templates := "SrcType := UInt" } EQ_Contact(in1 := #STATION_ALARM, in2 := 2)
      S_Coil( "DB440_MACHINE_ALARM_DECODING".ALARMS_UNIT_02.ST2_MEASURING.IS_SEOC_ALARMS )
   END_RUNG
   RUNG wire#w3
      { S7_Templates := "SrcType := UInt" } EQ_Contact(in1 := #STATION_ALARM, in2 := 3)
      S_Coil( "DB440_MACHINE_ALARM_DECODING".ALARMS_UNIT_02.ST3_CLADDING.IS_SEOC_ALARMS )
   END_RUNG
   RUNG wire#w3
      { S7_Templates := "SrcType := UInt" } EQ_Contact(in1 := #STATION_ALARM, in2 := 4)
      S_Coil( "DB440_MACHINE_ALARM_DECODING".ALARMS_UNIT_02.ST4_CLEANING.IS_SEOC_ALARMS )
   END_RUNG
   RUNG wire#w1
      { S7_Templates := "SrcType := UInt" } EQ_Contact(in1 := #UNIT_ALARM, in2 := 3)
      S_Coil( "DB440_MACHINE_ALARM_DECODING".ALARMS_UNIT_03.IS_SEOC_ALARMS )
   END_RUNG
   RUNG wire#w1
      { S7_Templates := "SrcType := UInt" } EQ_Contact(in1 := #UNIT_ALARM, in2 := 4)
      S_Coil( "DB440_MACHINE_ALARM_DECODING".ALARMS_UNIT_04.IS_SEOC_ALARMS )
   END_RUNG
   // the same network as SCL:
   // ENO of a box is taken as its EN; it also drops when the box reports an error
   #BRAKE.IS_SEOC_ALARMS := NOT (NOT #BLOCKED_ALARM AND NOT #UNBLOCKED_ALARM AND NOT #MAINTENANCE_UNBLOCKED_ALARM);
   IF #BRAKE.IS_SEOC_ALARMS THEN
       "DB440_MACHINE_ALARM_DECODING".GLOBAL_ALARMS_MACHINE.ALARM_DECODING := #DB_NUMBER;
   END_IF;
   #_w1 := #BRAKE.IS_SEOC_ALARMS AND (#UNIT_ALARM = 1);
   IF #_w1 AND (#STATION_ALARM = 0) THEN
       "DB440_MACHINE_ALARM_DECODING".ALARMS_UNIT_01.ST0_TRANSFER.IS_SEOC_ALARMS := TRUE;
   END_IF;
   IF #_w1 AND (#STATION_ALARM = 1) THEN
       "DB440_MACHINE_ALARM_DECODING".ALARMS_UNIT_01.ST1_LOAD_UNLOAD.IS_SEOC_ALARMS := TRUE;
   END_IF;
   IF #_w1 AND (#STATION_ALARM = 2) THEN
       "DB440_MACHINE_ALARM_DECODING".ALARMS_UNIT_01.ST2_SPARE.IS_SEOC_ALARMS := TRUE;
   END_IF;
   IF #_w1 AND (#STATION_ALARM = 3) THEN
       "DB440_MACHINE_ALARM_DECODING".ALARMS_UNIT_01.ST3_CLADDING.IS_SEOC_ALARMS := TRUE;
   END_IF;
   IF #_w1 AND (#STATION_ALARM = 4) THEN
       "DB440_MACHINE_ALARM_DECODING".ALARMS_UNIT_01.ST4_CLEANING.IS_SEOC_ALARMS := TRUE;
   END_IF;
   #_w2 := #BRAKE.IS_SEOC_ALARMS AND (#UNIT_ALARM = 2);
   IF #_w2 AND (#STATION_ALARM = 0) THEN
       "DB440_MACHINE_ALARM_DECODING".ALARMS_UNIT_02.ST0_TRANSFER.IS_SEOC_ALARMS := TRUE;
   END_IF;
   IF #_w2 AND (#STATION_ALARM = 1) THEN
       "DB440_MACHINE_ALARM_DECODING".ALARMS_UNIT_02.ST1_LOAD_UNLOAD.IS_SEOC_ALARMS := TRUE;
   END_IF;
   IF #_w2 AND (#STATION_ALARM = 2) THEN
       "DB440_MACHINE_ALARM_DECODING".ALARMS_UNIT_02.ST2_MEASURING.IS_SEOC_ALARMS := TRUE;
   END_IF;
   IF #_w2 AND (#STATION_ALARM = 3) THEN
       "DB440_MACHINE_ALARM_DECODING".ALARMS_UNIT_02.ST3_CLADDING.IS_SEOC_ALARMS := TRUE;
   END_IF;
   IF #_w2 AND (#STATION_ALARM = 4) THEN
       "DB440_MACHINE_ALARM_DECODING".ALARMS_UNIT_02.ST4_CLEANING.IS_SEOC_ALARMS := TRUE;
   END_IF;
   IF #BRAKE.IS_SEOC_ALARMS AND (#UNIT_ALARM = 3) THEN
       "DB440_MACHINE_ALARM_DECODING".ALARMS_UNIT_03.IS_SEOC_ALARMS := TRUE;
   END_IF;
   IF #BRAKE.IS_SEOC_ALARMS AND (#UNIT_ALARM = 4) THEN
       "DB440_MACHINE_ALARM_DECODING".ALARMS_UNIT_04.IS_SEOC_ALARMS := TRUE;
   END_IF;
END_REGION

REGION Network 30: ANY ACTIVE ALARM
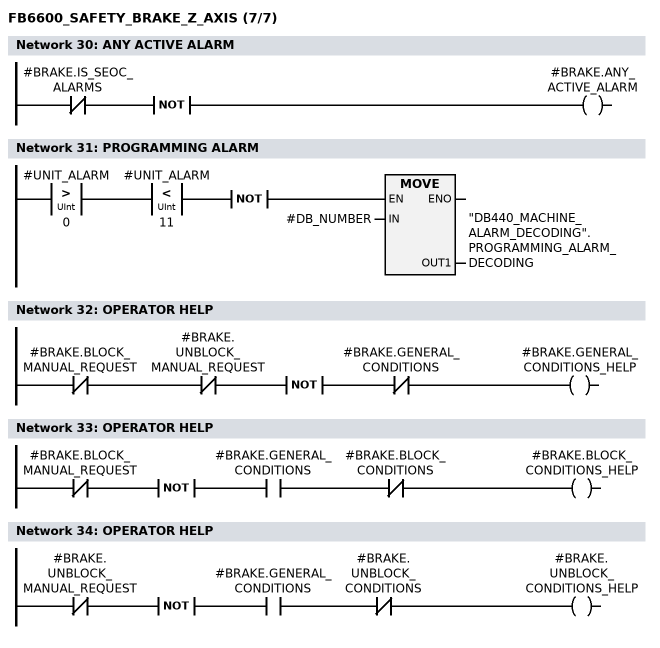
   RUNG wire#powerrail
      I_Contact( #BRAKE.IS_SEOC_ALARMS )
      Not()
      Coil( #BRAKE.ANY_ACTIVE_ALARM )
   END_RUNG
   // the same network as SCL:
   #BRAKE.ANY_ACTIVE_ALARM := NOT (NOT #BRAKE.IS_SEOC_ALARMS);
END_REGION

REGION Network 31: PROGRAMMING ALARM
   RUNG wire#powerrail
      { S7_Templates := "SrcType := UInt" } GT_Contact(in1 := #UNIT_ALARM, in2 := 0)
      { S7_Templates := "SrcType := UInt" } LT_Contact(in1 := #UNIT_ALARM, in2 := 11)
      Not()
      Move(in := #DB_NUMBER, out1 => "DB440_MACHINE_ALARM_DECODING".PROGRAMMING_ALARM_DECODING)
   END_RUNG
   // the same network as SCL:
   IF NOT ((#UNIT_ALARM > 0) AND (#UNIT_ALARM < 11)) THEN
       "DB440_MACHINE_ALARM_DECODING".PROGRAMMING_ALARM_DECODING := #DB_NUMBER;
   END_IF;
END_REGION

REGION Network 32: OPERATOR HELP
   RUNG wire#powerrail
      I_Contact( #BRAKE.BLOCK_MANUAL_REQUEST )
      I_Contact( #BRAKE.UNBLOCK_MANUAL_REQUEST )
      Not()
      I_Contact( #BRAKE.GENERAL_CONDITIONS )
      Coil( #BRAKE.GENERAL_CONDITIONS_HELP )
   END_RUNG
   // the same network as SCL:
   #BRAKE.GENERAL_CONDITIONS_HELP := NOT (NOT #BRAKE.BLOCK_MANUAL_REQUEST AND NOT #BRAKE.UNBLOCK_MANUAL_REQUEST) AND NOT #BRAKE.GENERAL_CONDITIONS;
END_REGION

REGION Network 33: OPERATOR HELP
   RUNG wire#powerrail
      I_Contact( #BRAKE.BLOCK_MANUAL_REQUEST )
      Not()
      Contact( #BRAKE.GENERAL_CONDITIONS )
      I_Contact( #BRAKE.BLOCK_CONDITIONS )
      Coil( #BRAKE.BLOCK_CONDITIONS_HELP )
   END_RUNG
   // the same network as SCL:
   #BRAKE.BLOCK_CONDITIONS_HELP := NOT (NOT #BRAKE.BLOCK_MANUAL_REQUEST) AND #BRAKE.GENERAL_CONDITIONS AND NOT #BRAKE.BLOCK_CONDITIONS;
END_REGION

REGION Network 34: OPERATOR HELP
   RUNG wire#powerrail
      I_Contact( #BRAKE.UNBLOCK_MANUAL_REQUEST )
      Not()
      Contact( #BRAKE.GENERAL_CONDITIONS )
      I_Contact( #BRAKE.UNBLOCK_CONDITIONS )
      Coil( #BRAKE.UNBLOCK_CONDITIONS_HELP )
   END_RUNG
   // the same network as SCL:
   #BRAKE.UNBLOCK_CONDITIONS_HELP := NOT (NOT #BRAKE.UNBLOCK_MANUAL_REQUEST) AND #BRAKE.GENERAL_CONDITIONS AND NOT #BRAKE.UNBLOCK_CONDITIONS;
END_REGION
END_FUNCTION_BLOCK
